TYPE ST_AutomaticExtractionValues :
STRUCT
	elapsedTime : TIME;
	currentTimer : TIME;
	timeVisible : BOOL;
END_STRUCT
END_TYPE

(* stored: Version 1.1.0.1, ProductVersion 3.1.4024.9
   DUT ST_AutomaticExtractionValues: Id {4a423156-e99e-429d-98a3-547a859b5d8a} *)
